(*********************************** G.D S.p.A. - Technical Department ***********************************
============= PROGRAM INFO ============
FOLDER:             TBD
MACHINES INVOLVED:  TBD 

============= DESCRIPTION =============
Machine declaration

============= REVISIONS ===============
Date		Version	 	Author      	Description             
----------	-------		------------  	--------------------------------------------
2019/03/27 	0000.00	 	CEC 			Creation of the PRG

**********************************************************************************************************)

TYPE csp_customerInterfaces_casePackerStFault :
STRUCT
	
	Main:				BOOL;				(*$H_R desc := Main machine is faulted; $*)
	CaseBlanks:			BOOL;				(*$H_R desc := Local case blank supply system is faulted; $*)
															
END_STRUCT
END_TYPE

(* stored: Version 1.1.0.1, ProductVersion 3.1.4024.3
   DUT csp_customerInterfaces_casePackerStFault: Id {f4e16dcf-7f38-4817-b66e-3eab1df235a6} *)
